FUNCTION_BLOCK ReadEncSpeed
VAR_INPUT
	input1:BOOL;
END_VAR
VAR_OUTPUT
	RealSpeed:REAL;
END_VAR
VAR
	ver1	:MC_ReadActualVelocity;
END_VAR

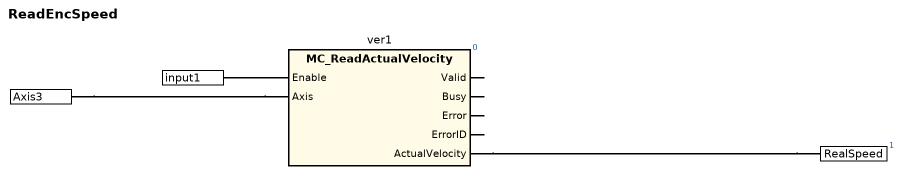
ver1(Enable := input1, Axis := Axis3); // MC_ReadActualVelocity
RealSpeed := ver1.ActualVelocity;

END_FUNCTION_BLOCK

(* stored: Version 1.1.0.1, ProductVersion 3.1.4024.12
   POU ReadEncSpeed: Id {5313854b-9c9a-44b2-a8ea-d6ee320775a6}, SpecialFunc None *)
